(* CODESYS project projekt-inzynierka-final.ecp

Project tree, tasks and I/O mapping:
  GenericDummyMasterDevice : Generic Master, WAGO, order no. None, version 1.0.0.0
  PFC200_CS_2ETH_RS : 750-8202 PFC200 2ETH RS, WAGO, order no. 0750-8202, version 1.4.1.22
    application Application
      libraries: ; WagoAppPlcModbus, * (WAGO); WagoAppCom, * (WAGO)
      task PLC_Task (cyclic, interval t#10ms, priority 14) calls PLC_PRG, pracaCykliczna, analizator, zapisDanychPomiarowychProgram
      task VISU_TASK (cyclic, interval 100 ms, priority 15) calls VisuElems.Visu_Prg
      program PLC_PRG [ST]
      program analizator [ST]
      function dostosowanieCO [ST]
      function dostosowanieO2 [ST]
      program pracaCykliczna [LD]
      function word2real [ST]
      global variables GVL
      visualisation PLC_VISU
      program zapisDanychPomiarowychProgram [CFC]
    DeviceAdapter
    Kbus : Kbus, WAGO, version 1.3.0.0
        unmapped channels: K-BUS diagnostics
      RS_232_RS_485_Interface_adjustable : 0750-0652, WAGO, order no. 0750-0652, version 0.0.0.22
          settings: K-BUS Module slot index = 1
          unmapped channels: _INPUTCHANNEL, _OUTPUTCHANNEL
        DeviceAdapter
      _4_AO_0_10V_DC : 0750-0559, WAGO, order no. 0750-0559, version 0.0.0.11
          settings: K-BUS Module slot index = 2
          output przep3 : WORD  // _QW 1
          output przep2 : WORD  // _QW 2
          output przep1 : WORD  // _QW 3
          unmapped channels: _QW 4
        DeviceAdapter
      _4_AI_4_20mA_s_e : 0750-0455, WAGO, order no. 0750-0455, version 0.0.0.10
          settings: K-BUS Module slot index = 3
          unmapped channels: _IW 1, _IW 2, _IW 3, _IW 4
        DeviceAdapter
      _2_AI_Thermocouple_K_Diag : 0750-0469, WAGO, order no. 0750-0469, version 0.0.0.7
          settings: K-BUS Module slot index = 4
          input  ai_pttk_01 : INT  // _IINT 1
          unmapped channels: _IINT 2
        DeviceAdapter
    MODBUS
      MODBUS : MODBUS, WAGO, order no. n/a, version 1.1.1.13
    Serial
      COM1 : COM1, WAGO, version 0.0.0.19
  libraries: VisuSymbols, 3.5.8.0 (System); WagoVisuIcons, 1.0.0.0 (WAGO); WagoAppDatalogger, 1.0.0.7 (WAGO)
  text list GlobalTextList
*)

// PFC200_CS_2ETH_RS/Application/GVL
{attribute 'qualified_only'}
VAR_GLOBAL
	przepustnica1: WORD :=100; //Do przypisania z hardware - przepustnica1 - od CO
	przepustnica2: WORD := 50;//Do przpisania z hardware - przepustnica2 - Od O2
	pomiarTemp: REAL; //Do przypisania z hardware Temp spalin
	
	normaCO : REAL := 900; //Maksymalna wartość CO którą chcemy uzyskiwać [ppm]
	normaO2 : REAL := 13; //Wartosc O2 którą chcemy utrzymywać [%]
	
	deltaT: TIME := T#10S; //Czas pomiędzy pobieraniem danych do wyznaczenia trendu
	
	przepMIN: WORD := 0; //Minimalne otwarcie przepustnicy [%]
	przepMAX: WORD := 100; //Maksymalne otwarcie przepustnicy [%]
	deltaPrzep: WORD := 5; //Krok otwarcia przepustnicy [%]
	
	timeTrigger: BOOL := FALSE; //Trigger z licznika, odpala się co deltaT
	timeTriggerReset: BOOL := FALSE; //Reset timera 0->1 start timera, 1->0 reset timera
	
	//Pomiary z analizatora spalin
	pomiarCO: REAL;
	pomiarO2: REAL;
	pomiarCO2: REAL;
	pomiarNO: REAL;
	pomiarNO2: REAL;
	pomiarNOx: REAL;
	pomiarSO2: REAL;
	
	wartosci: ARRAY[1..MAX_CHANNELS] OF REAL := [
		GVL.pomiarCO, 
		GVL.pomiarO2, 
		WORD_TO_REAL(GVL.przepustnica1), 
		WORD_TO_REAL(GVL.przepustnica2), 
		GVL.normaCO,
		GVL.normaO2,
		GVL.pomiarNOx,
		GVL.pomiarSO2,
		GVL.pomiarCO2,
		GVL.pomiarTemp
		];
END_VAR

// PFC200_CS_2ETH_RS/Application/PLC_PRG
PROGRAM PLC_PRG
VAR
	//Pomiary danych do stworzenia trendów 
	spalinyCO_pomiar1: REAL := 0; //Pomiar 1. CO
	spalinyO2_pomiar1: REAL := 0; //Pomiar 1. O2
	spalinyTemp_pomiar1: REAL := 0; //Pomiar 1. Temp Spalin
	
	spalinyCO_pomiar2: REAL := 0; //Pomiar 2. CO
	spalinyO2_pomiar2: REAL := 0; //Pomiar 2. O2
	spalinyTemp_pomiar2: REAL := 0; //Pomiar 2. Temp Spalin
	
	spalinyCO_pomiar3: REAL := 0; //Pomiar 3. CO
	spalinyO2_pomiar3: REAL := 0; //Pomiar 3. O2
	spalinyTemp_pomiar3: REAL := 0; //Pomiar 3. Temp Spalin
	
	Prio: BOOL := TRUE; //Priorytet dla dostosowanieO2 dla przepustnicy3
	zbocz_o: R_TRIG;
	zbocze: BOOL;
END_VAR

zbocz_o(CLK:=GVL.timeTrigger, Q=> zbocze);
GVL.pomiarTemp := INT_TO_REAL(ai_pttk_01)/10;
IF zbocze THEN
	IF spalinyCO_pomiar1 = 0 THEN
		spalinyCO_pomiar1 := GVL.pomiarCO;
		spalinyO2_pomiar1 := GVL.pomiarO2;
		spalinyTemp_pomiar1 := GVL.pomiarTemp;
	ELSIF spalinyCO_pomiar2 = 0 THEN
		spalinyCO_pomiar2 := GVL.pomiarCO;
		spalinyO2_pomiar2 := GVL.pomiarO2;
		spalinyTemp_pomiar2 := GVL.pomiarTemp;
	ELSIF spalinyCO_pomiar3 = 0 THEN
		spalinyCO_pomiar3 := GVL.pomiarCO;
		spalinyO2_pomiar3 := GVL.pomiarO2;
		spalinyTemp_pomiar3 := GVL.pomiarTemp;
		Prio := dostosowanieCO(P1:=spalinyCO_pomiar1, P2:=spalinyCO_pomiar2, P3:=spalinyCO_pomiar3);
		dostosowanieO2(P1:=spalinyO2_pomiar1, P2:=spalinyO2_pomiar2, P3:=spalinyO2_pomiar3, Prio:=Prio);
		
		//Zerowanie wyników
		spalinyCO_pomiar1 := 0;
		spalinyCO_pomiar2 := 0;
		spalinyCO_pomiar3 := 0;
		Prio := TRUE;
	END_IF
	przep1:=24575-GVL.przepustnica1*164;
	przep2:=24575-GVL.przepustnica2*164;
END_IF
GVL.wartosci[1] := GVL.pomiarCO;
GVL.wartosci[2] := GVL.pomiarO2;
GVL.wartosci[3] := WORD_TO_REAL(GVL.przepustnica1);
GVL.wartosci[4] := WORD_TO_REAL(GVL.przepustnica2);
GVL.wartosci[5] := GVL.normaCO;
GVL.wartosci[6] := GVL.normaO2;
GVL.wartosci[7] := GVL.pomiarNOx;
GVL.wartosci[8] := GVL.pomiarSO2;
GVL.wartosci[9] := GVL.pomiarCO2;
GVL.wartosci[10] := GVL.pomiarTemp;

END_PROGRAM

// PFC200_CS_2ETH_RS/Application/dostosowanieCO
FUNCTION dostosowanieCO : BOOL
VAR_INPUT
	P1: REAL;
	P2: REAL;
	P3: REAL;
END_VAR
VAR
	realPrzepMIN: WORD := GVL.przepMIN;//(GVL.przepMIN/100)*65535; //Minimalne otwarcie przepustnicy
	realPrzepMAX: WORD := GVL.przepMAX; //(GVL.przepMAX/100)*65535; //Maksymalne otwarcie przepustnicy 
	realDeltaPrzep: WORD := GVL.deltaPrzep; //Krok otwarcia przepustnicy
	realNormaCO : REAL := GVL.normaCO; //Maksymalna wartość CO którą chcemy uzyskiwać [?]
END_VAR

IF P1>realNormaCO OR P2>realNormaCO OR P3>realNormaCO THEN
	IF P1 <= P2 THEN
		IF P2 <= P3 THEN
			IF GVL.przepustnica1+realDeltaPrzep < realPrzepMAX THEN
				GVL.przepustnica1:=GVL.przepustnica1+realDeltaPrzep;
				dostosowanieCO := FALSE;
			END_IF		
		END_IF
	END_IF
ELSE
	IF P1 > P2 THEN
		IF P2 > P3 THEN
			IF GVL.przepustnica1-realDeltaPrzep > realPrzepMIN THEN
				GVL.przepustnica1:=GVL.przepustnica1-GVL.deltaPrzep;
				dostosowanieCO := FALSE;
			END_IF	
		END_IF
	END_IF
END_IF

END_FUNCTION

// PFC200_CS_2ETH_RS/Application/dostosowanieO2
FUNCTION dostosowanieO2 : BOOL
VAR_INPUT
	P1: REAL;
	P2: REAL;
	P3: REAL;
	Prio: BOOL;
END_VAR
VAR
	realPrzepMIN: WORD := GVL.przepMIN; //Minimalne otwarcie przepustnicy
	realPrzepMAX: WORD := GVL.przepMAX; //Maksymalne otwarcie przepustnicy
	realDeltaPrzep: WORD; //Krok otwarcia przepustnicy
	realNormaO2 : REAL := GVL.normaO2; //Wartosc O2 którą chcemy utrzymywać [?]
END_VAR

IF P1 <> realNormaO2 OR P2 <> realNormaO2 OR P3 <> realNormaO2 THEN
	IF P1 < realNormaO2 OR P2 < realNormaO2 OR P3 < realNormaO2 THEN
		IF GVL.przepustnica2+realDeltaPrzep < realPrzepMAX THEN
			GVL.przepustnica2:=GVL.przepustnica2+GVL.deltaPrzep;	
		END_IF
	ELSIF P1 > realNormaO2 OR P2 > realNormaO2 OR P3 > realNormaO2 THEN
		IF GVL.przepustnica2-realDeltaPrzep > realPrzepMIN THEN
			GVL.przepustnica2:=GVL.przepustnica2-GVL.deltaPrzep;
		ELSE
			IF GVL.przepustnica1-realDeltaPrzep > realPrzepMIN THEN
				GVL.przepustnica1:=GVL.przepustnica1-GVL.deltaPrzep;
			END_IF
		END_IF	
	END_IF
END_IF

END_FUNCTION

// PFC200_CS_2ETH_RS/Application/pracaCykliczna
PROGRAM pracaCykliczna
VAR
	T01: TON;
	T02: TOF;
END_VAR

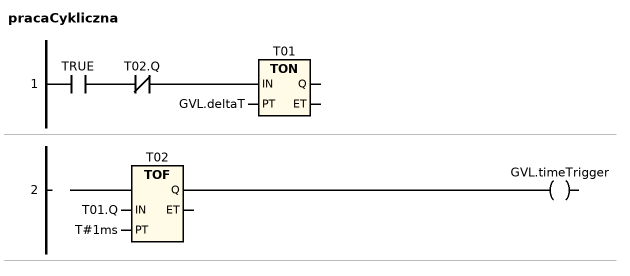
// NETWORK 1
T01(IN := TRUE AND NOT T02.Q, PT := GVL.deltaT); // TON

// NETWORK 2
T02(IN := T01.Q, PT := T#1ms); // TOF
GVL.timeTrigger := T02.Q;

END_PROGRAM

// PFC200_CS_2ETH_RS/Application/analizator
PROGRAM analizator
VAR
	start: BOOL;
	polaczono: BOOL;
	zapytanie: typMbQuery;
	odpowiedz: typMbResponse;
	MODBUS_EXTENDED_MASTER_1: FbMbMasterSerial;
	dane: ARRAY [0..124] OF WORD;
	status: WagoSysErrorBase.FbResult;
	adresSL: WORD;
	TON_generator: TON;
END_VAR

MODBUS_EXTENDED_MASTER_1(
	xConnect:=TRUE , 
	xTrigger:=start,
	I_PORT:=RS_232_RS_485_Interface_adjustable,
	udiBaudrate:= 9600,
	usiDataBits:= 8, 
	eParity:=eTTYParity.Even , 
	eStopBits:= eTTYStopBits.one, 
	ePhysical:= RS232,
	eFrameType:= RTU,
	utQuery:= zapytanie,
	utResponse:=odpowiedz,
	xIsConnected=>polaczono,
	tTimeOut:=T#1S,
	);

zapytanie.bUnitId:=1;
zapytanie.uiReadAddress:=20;
zapytanie.uiReadQuantity:=20;
zapytanie.bFunctionCode:=3;

TON_generator(IN:=NOT TON_generator.Q AND NOT start  , PT:=T#1S , Q=> , ET=> );
start S= TON_generator.Q;
IF polaczono THEN
	dane:=odpowiedz.awData;
	GVL.pomiarO2:= word2real(dane[1],dane[0]);
	GVL.pomiarCO2:= (word2real(dane[3],dane[2]));
	GVL.pomiarCO:= word2real(dane[5],dane[4])*((8/(21-GVL.pomiarO2)));
	GVL.pomiarNO:= word2real(dane[7],dane[6]);
	GVL.pomiarNO2:= word2real(dane[9],dane[8]);
	GVL.pomiarNOx:= word2real(dane[11],dane[10]);
	GVL.pomiarSO2:= word2real(dane[13],dane[12]);
END_IF

END_PROGRAM

// PFC200_CS_2ETH_RS/Application/word2real
FUNCTION word2real : REAL
VAR_INPUT
	w2: WORD;
	w1: WORD;
END_VAR
VAR
	wsk: POINTER TO ARRAY[1..2] OF WORD;
	tmp: REAL;
END_VAR

wsk:=ADR(tmp);
wsk^[2]:=w1;
wsk^[1]:=w2;
word2real:=tmp;

END_FUNCTION

// PFC200_CS_2ETH_RS/Application/zapisDanychPomiarowychProgram
PROGRAM zapisDanychPomiarowychProgram
VAR
	privEvent: BOOL := TRUE;	

	kanal1: typChannelConfig := (
	xChannelExists:= TRUE,  
	sChannelName:= 'PomiarCO', 
	sUnit:= 'ppm');
	
	kanal2: typChannelConfig := (
	xChannelExists:= TRUE,  
	sChannelName:= 'PomiarO2', 
	sUnit:= '%');
	
	kanal3: typChannelConfig := (
	xChannelExists:= TRUE,  
	sChannelName:= 'Przepustnica1', 
	sUnit:= '%');
	
	kanal4: typChannelConfig := (
	xChannelExists:= TRUE,  
	sChannelName:= 'Przepustnica2', 
	sUnit:= '%');
	
	kanal5: typChannelConfig := (
	xChannelExists:= TRUE,  
	sChannelName:= 'NormaCO', 
	sUnit:= 'ppm');
	
	kanal6: typChannelConfig := (
	xChannelExists:= TRUE,  
	sChannelName:= 'NormaO2', 
	sUnit:= '%');
	
	kanal7: typChannelConfig := (
	xChannelExists:= TRUE,  
	sChannelName:= 'PomiarNOx', 
	sUnit:= 'ppm');
	
	kanal8: typChannelConfig := (
	xChannelExists:= TRUE,  
	sChannelName:= 'PomiarSO2', 
	sUnit:= 'ppm');
	
	kanal9: typChannelConfig := (
	xChannelExists:= TRUE,  
	sChannelName:= 'PomiarCO2', 
	sUnit:= '%');
	
	kanal10: typChannelConfig := (
	xChannelExists:= TRUE,  
	sChannelName:= 'PomiarTemp', 
	sUnit:= 'stC');
	
	kanaly: ARRAY[1..MAX_CHANNELS] OF typChannelConfig := [kanal1, kanal2, kanal3, kanal4, kanal5, kanal6, kanal7, kanal8, kanal9, kanal10];
	
	dataLoggingConfig: typConfigDatalogger := (
	bDatalogger_type:= 1, 
	xAppendDate:= TRUE, 
	xCyclicLogging:= TRUE, 
	bInterval:= 3, 
	sFilename:= 'dane_pomiarowe.csv', 
	sPath:= '/home/codesys_root',  
	atypChannelConfig:= kanaly);
	dataLogger: FbDatalogger;
END_VAR

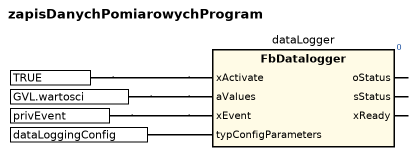
dataLogger(
    xActivate := TRUE,
    aValues := GVL.wartosci,
    xEvent := privEvent,
    typConfigParameters := dataLoggingConfig); // FbDatalogger

END_PROGRAM

// PFC200_CS_2ETH_RS/Application/PLC_VISU
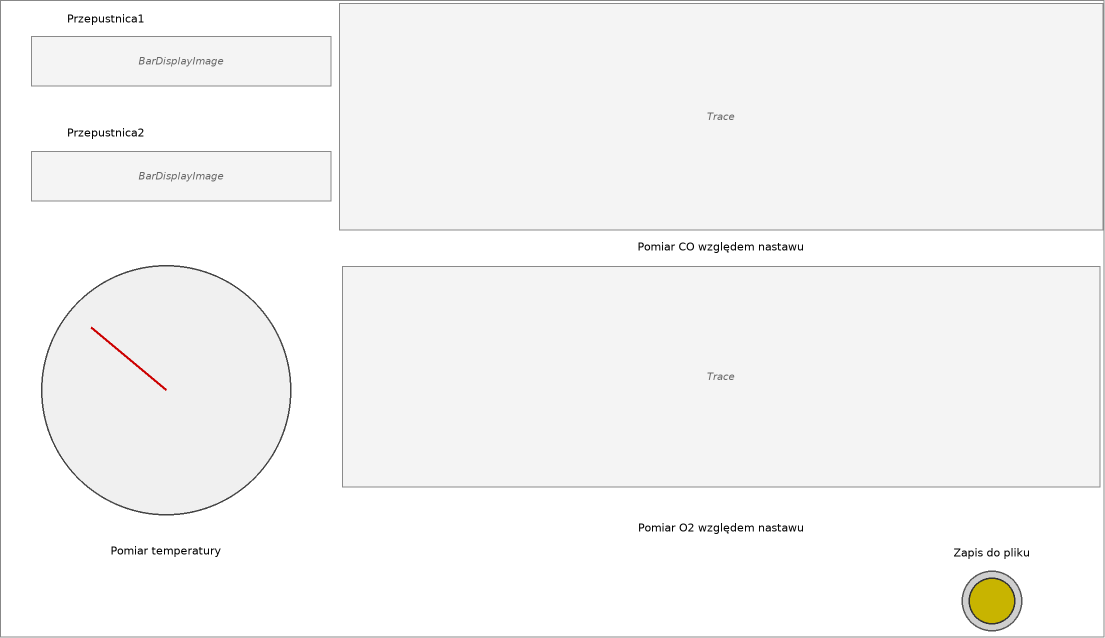
VISUALIZATION PLC_VISU  // 1105x638
    BarDisplayImage (31,36 300x50), value: GVL.przepustnica1, style: BarDisplayImage-Gray, scale format: %.1f, scale 0..100
    BarDisplayImage (31,151 300x50), value: GVL.przepustnica2, style: BarDisplayImage-Gray, scale format: %.1f, scale 0..100
    Label (31,4 150x30), "Przepustnica1"
    Label (31,118 150x30), "Przepustnica2"
    Label (593,232 256x30), "Pomiar CO względem nastawu"
    Trace (342,266 758x221)
    Label (593,513 256x30), "Pomiar O2 względem nastawu"
    Lamp1 (957,566 70x70), variable: zapisDanychPomiarowychProgram.dataLogger._xFileOk, style: Lamp-Lamp1-Yellow
    Meter360 (41,265 250x250), value: GVL.pomiarTemp, style: Meter-Meter360-Gray, scale format: %.1f, scale 0..500
    Label (38,536 256x30), "Pomiar temperatury"
    Trace (339,3 764x227)
    Label (917,538 150x30), "Zapis do pliku"
END_VISUALIZATION
